FUNCTION_BLOCK FB_SlaveArmCheck
VAR_INPUT
END_VAR
VAR_OUTPUT
END_VAR
VAR
	// final arm error flag
	m_armErrFlag :ARRAY[1..g_sArmNum] OF BOOL:=[4(FALSE)];
	
	// cartesian pose error flag
	m_cartPoseErrFlag :ARRAY[1..g_sArmNum] OF BOOL;
	m_cartPoseErrCounts:ARRAY[1..g_sArmNum] OF INT;
	m_cartPosErr :ARRAY[1..g_sArmNum] OF Vec3d;	// cartesian position error
	m_cartOriErr:ARRAY[1..g_sArmNum] OF  Vec3d;	// cartesian rotation angle (angle  * axis)
	
	// joint control error flag
	m_jntCtrlErrFlag :ARRAY[1..g_sArmNum] OF Vec8b;
	m_jntCtrlErrCounts :ARRAY[1..g_sArmNum] OF Vec8i;
	m_jntCtrlErr:ARRAY[1..g_sArmNum]  OF Vec8d;		// joint position control error
	
	// joint encoder error flag
	m_jntEncErrFlag :ARRAY[1..g_sArmNum] OF Vec8b;
	m_jntEncErrCounts :ARRAY[1..g_sArmNum] OF Vec8i ;
	m_jntEncErr:ARRAY[1..g_sArmNum]  OF Vec8d;		// motor and joint encoder error
	
	// joint velocity error flag
	m_jntVelErrFlag :ARRAY[1..g_sArmNum] OF Vec8b;
	m_jntVelErrCounts :ARRAY[1..g_sArmNum] OF Vec8i;
	
	// joint position limit error flag
	m_jntLimitErrFlag :ARRAY[1..g_sArmNum] OF Vec8b;
	m_jntLimitErrCounts :ARRAY[1..g_sArmNum] OF Vec8i;

END_VAR

METHOD check : BOOL
VAR_IN_OUT CONSTANT
	i_slaveStatus : ST_SlaveStatus;
	i_slaveJointData :ST_SlaveJointData;
END_VAR
VAR_OUTPUT
	o_errorFlag :ARRAY[1..g_sArmNum] OF BOOL ;
END_VAR

VAR
	i ,j:INT ;
END_VAR
// calculate error
FOR i:=1 TO g_sArmNum DO 
	// stop check if arm is already in error state
	IF m_armErrFlag[i] OR i_slaveStatus.m_armState[i]=SlaveArmState_Error THEN 
		CONTINUE;
	END_IF
	
	// only check cartesion pose error in master-slave mode and within joint limit
	m_cartPoseErrFlag[i]:=FALSE;
	IF  SlaveArmState_MasterSlave = i_slaveStatus.m_armState[i] THEN 
		m_cartPoseErrFlag[i]:=poseErrCheck(i_slaveStatus.m_cmdArmPose[i],  i_slaveStatus.m_curArmPose[i],
											m_cartPoseErrCounts[i], m_cartPosErr[i], m_cartOriErr[i]);
	END_IF
	
	// joint control error
	m_jntCtrlErrFlag[i]:=jntCtrlErrCheck(i_slaveJointData.m_cmdJntPos[i], i_slaveJointData.m_curJntPos[i],
										m_jntCtrlErrCounts[i], m_jntCtrlErr[i]);
	
	// encoder error
	m_jntEncErrFlag[i]:=jntEncErrCheck(i_slaveJointData.m_curMotorPos[i], i_slaveJointData.m_curLinkPos[i],
										m_jntEncErrCounts[i], m_jntEncErr[i]);
										
	// joint limit error
	m_jntLimitErrFlag[i]:=jntLimitErrCheck(i_slaveJointData.m_curJntPos[i],m_jntLimitErrCounts[i]);
										
	// final arm error status check
	IF  m_cartPoseErrFlag[i] THEN
		m_armErrFlag[i]:=TRUE;
		CONTINUE;
	END_IF
	
	FOR j:=1 TO g_sJntNum DO 
		IF m_jntCtrlErrFlag[i][j] OR m_jntEncErrFlag[i][j] OR m_jntVelErrFlag[i][j] OR m_jntLimitErrFlag[i][j] THEN
			m_armErrFlag[i]:=TRUE;
			EXIT;
		END_IF
	END_FOR
	
END_FOR

o_errorFlag:=m_armErrFlag;
END_METHOD

METHOD jntCtrlErrCheck : Vec8b
VAR_INput
	i_cmdJntPos : Vec8d;
	i_curJntPos : Vec8d;
END_VAR
VAR_IN_OUT
	r_errCount:Vec8i;
	r_jntCtrlErr :Vec8d;
END_VAR

VAR
	i :INT;
	err:Vec8d;
END_VAR
vecSub(i_cmdJntPos,i_curJntPos,  err);
r_jntCtrlErr:=err;

// joint error check
//NOTE: only check the first three joints.
FOR i:=1 TO 3 DO 
	IF  ABS(r_jntCtrlErr[i]) > g_slaveMaxJntCtrlErr[i] THEN
		r_errCount[i]:=r_errCount[i]+1;
	ELSE
		r_errCount[i] :=0;	
	END_IF
	jntCtrlErrCheck[i]:= r_errCount[i]>=g_faultTriggerCounts;
END_FOR
END_METHOD

METHOD jntEncErrCheck : Vec8b
VAR_INput
	i_motorJntPos : Vec8d;
	i_linkJntPos : Vec8d;
END_VAR
VAR_IN_OUT
	r_errCount:Vec8i;
	r_jntEncErr :Vec8d;
END_VAR

VAR
	i :INT;
	err:Vec8d;
END_VAR
vecSub(i_motorJntPos,i_linkJntPos,  err);
r_jntEncErr:=err;

// joint error check
FOR i:=1 TO g_sJntNum DO 
	IF  ABS(r_jntEncErr[i]) > g_slaveMaxJntCtrlErr[i] THEN
		r_errCount[i]:=r_errCount[i]+1;
	ELSE
		r_errCount[i] :=0;
	END_IF
	jntEncErrCheck[i]:= r_errCount[i]>=g_faultTriggerCounts;
END_FOR

// NOTE: power box joints are easy to trigger encoder error during instrument mount, so this part is diabled now
FOR i:=4 TO g_sJntNum DO
	jntEncErrCheck[i] := false;
END_FOR
END_METHOD

METHOD jntLimitErrCheck : Vec8b
VAR_INput
	i_curJntPos : Vec8d;
END_VAR
VAR_IN_OUT
	r_errCount:Vec8i;
END_VAR

VAR
	i :INT;
END_VAR
// joint limit check
//NOTE: only check the first three joints.
FOR i:=1 TO 3 DO 
	IF  i_curJntPos[i] > GVL_SlaveMotorParameters.g_maxJntPos[i] + g_slaveJntPosLimitBuffer[i] OR
		i_curJntPos[i] < GVL_SlaveMotorParameters.g_minJntPos[i] - g_slaveJntPosLimitBuffer[i] THEN
		r_errCount[i]:=r_errCount[i]+1;
	ELSE
		r_errCount[i] :=0;	
	END_IF
	jntLimitErrCheck[i]:= r_errCount[i]>=g_faultTriggerCounts;
END_FOR
END_METHOD

METHOD poseErrCheck : BOOL
VAR_INPUT
	i_cmdPose : ST_Frame;
	i_curPose :ST_Frame;
END_VAR
VAR_IN_OUT
	r_errCount:INT;
	r_posErr :Vec3d;
	r_oriErr :Vec3d;
END_VAR

VAR
	posErr,oriErr:Vec3d;
	matT,rotErr:Mat3d;
	errAngle :LREAL;
	errAxis :Vec3d;
END_VAR
vecSub(i_cmdPose.m_pos, i_curPose.m_pos,posErr);
r_posErr:=posErr;

matTranspose(i_cmdPose.m_rot, matT);
matMultiply(matT,i_curPose.m_rot, rotErr);
rot2AngAxis(rotErr, angle=>errAngle, axis=>errAxis);
vecMultiNum(errAxis, errAngle,oriErr);
r_oriErr:=oriErr;
	
IF  norm(posErr)>g_maxCartPosErr OR norm(oriErr)> g_maxCartOriErr THEN
	r_errCount:= r_errCount +1;
ELSE 
	r_errCount:=0;
END_IF
poseErrCheck:= r_errCount >= g_faultTriggerCounts;
END_METHOD

END_FUNCTION_BLOCK

(* stored: Version 1.1.0.1, ProductVersion 3.1.4024.12
   POU FB_SlaveArmCheck: Id {7fa43d5a-568e-4b76-ad81-6c5cf7c4ee74}, SpecialFunc None
   Method check: Id {321cd4e5-6c66-4065-8a9a-a49a4a7544f4}
   Method jntCtrlErrCheck: Id {f2b82bf6-f8b5-4f0c-98ca-679940c1f1fb}
   Method jntEncErrCheck: Id {31ef1a61-be8a-4cf4-8816-44c2de3e927b}
   Method jntLimitErrCheck: Id {a4da3795-73c8-472d-94c8-3533763f2a83}
   Method poseErrCheck: Id {9fe210b5-ecf0-4498-8364-258d193de1ff} *)
